{attribute 'GeneratedUsingTerminal: KL9210'}
{attribute addProperty BoxType "KL9210"}
{attribute addProperty Id "Channel_1AT %I*Channel_64AAC8C70"}
{attribute addProperty CRC "2347652594"}
{attribute addProperty Size "0"}
TYPE KL9210_8BEE55F2 :
STRUCT
	{attribute addProperty Name "Channel_1"}
	Channel_1 : Channel_64AAC8C7;
END_STRUCT
END_TYPE

(* stored: Version 1.2.0.0, ProductVersion 3.1.4024.9
   DUT KL9210_8BEE55F2: Id {96af066a-8b81-4d8f-a2ca-30e5f2476917} *)
